FUNCTION_BLOCK E_D_FF (* Data latch (d) flip flop *)
  (* Standard: 61499-1 Annex A; Description: Copyright (c) 2017 fortiss GmbH This program and the accompanying materials are made available under the terms of the Eclipse Public License 2.0 which is available at https://www.eclipse.org/legal/epl-2.0/ SPDX-License-Identifier: EPL-2.0 *)
  (* Version 1.0, 2017-09-22, Alois Zoitl, fortiss GmbH, initial API and implementation and/or initial documentation *)
  (* Version 3.0, 2025-04-14, Patrick Aigner, changed package *)
  PACKAGE iec61499::events;
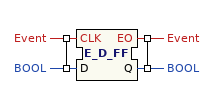
  EVENT_INPUT
    CLK WITH D; (* Clock *)
  END_EVENT
  EVENT_OUTPUT
    EO WITH Q; (* Triggered if clock results in a change of Q *)
  END_EVENT
  VAR_INPUT
    D : BOOL; (* Value to latch *)
  END_VAR
  VAR_OUTPUT
    Q : BOOL; (* Latched value *)
  END_VAR
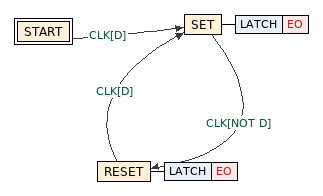
  EC_STATES
    START; (* Initial State *)
    SET : LATCH -> EO; (* Initialization *)
    RESET : LATCH -> EO;
  END_STATES
  EC_TRANSITIONS
    START TO SET := CLK[D];
    SET TO RESET := CLK[NOT D];
    RESET TO SET := CLK[D];
  END_TRANSITIONS
  ALGORITHM LATCH IN ST: (* new algorithm *)
Q := D;
  END_ALGORITHM
END_FUNCTION_BLOCK
